TYPE U_TICKET_LIST_DATA_INPUT :
UNION
  stData              : ST_LIST_NODE_DATA;
  byData   AT %I*     : ARRAY[1..SIZEOF(ST_LIST_NODE_DATA)] OF BYTE;
END_UNION
END_TYPE

(* stored: Version 1.1.0.1, ProductVersion 3.1.4026.13
   DUT U_TICKET_LIST_DATA_INPUT: Id {751a5806-4ac7-4ff3-b26c-58595e100566} *)
